// TwinCAT 3 PLC project PLC1
// ProgramVersion: 3.1.4023.0
// libraries:
//   Tc2_Standard, * (Beckhoff Automation GmbH)
//   Tc2_System, * (Beckhoff Automation GmbH)
//   Tc3_Module, * (Beckhoff Automation GmbH)
// project tree:
//   / PlcTask.TcTTO
//   POUs/ MAIN.TcPOU
// real-time tasks:
//   TASK PlcTask: cycle T#10ms, priority 20, ADS port 350
// I/O:
//   DEVICE Device 1 (EtherCAT) (disabled), AmsNetId 5.25.243.28.2.1
//   DEVICE Device 3 (NOV-DP-RAM)
//     Box 1 (Retain Handler)
// variable links:
//   PLC1/PLC1 Instance <-> Device 3 (NOV-DP-RAM)/Box 1 (Retain Handler)
//     PlcTask Retains/MAIN.arrTest <-> Retains/MAIN.arrTest_[851]
//     PlcTask Retains/MAIN.arrTest2 <-> Retains/MAIN.arrTest2_[851]
//     PlcTask Retains/MAIN.nivelBomba <-> Retains/MAIN.nivelBomba_[851]
//     PlcTask Retains/MAIN.x <-> Retains/MAIN.x_[851]
//     PlcTask Retains/MAIN.y <-> Retains/MAIN.y_[851]
//     PlcTask Retains/MAIN.z <-> Retains/MAIN.z_[851]

CONFIGURATION PLC1
    RESOURCE PLC ON TwinCAT3
        TASK PlcTask(INTERVAL := T#10ms, PRIORITY := 20);
        PROGRAM MAIN WITH PlcTask : MAIN;
    END_RESOURCE
END_CONFIGURATION

// ---- POUs/MAIN.TcPOU
PROGRAM MAIN
VAR RETAIN
	x	: UINT;
	y	: UINT;
	z	: UINT;
	arrTest : ARRAY[0..49] OF INT;
	arrTest2 : ARRAY[0..49] OF INT;
	
	nivelBomba : INT;
END_VAR

VAR
	i	: INT;
END_VAR

(*
FOR i := 0  TO 49 BY 1 DO
	IF ((i MOD 2) <> 0) THEN
		arrTest[i] 		:= i + 1969;
		arrTest2[i] 	:= arrTest[i+1];
	ELSE
		arrTest[i] 		:= i - 1998;
		arrTest2[i] 	:= arrTest[i+1];
	END_IF;
END_FOR;
*)

END_PROGRAM
